FUNCTION_BLOCK FB_Observer_USINT EXTENDS FB_AbstractObserver
VAR
    _nVal:              USINT;
END_VAR

METHOD FB_init : BOOL
VAR_INPUT
	bInitRetains : BOOL; // if TRUE, the retain variables are initialized (warm start / cold start)
	bInCopyCode : BOOL;  // if TRUE, the instance afterwards gets moved into the copy code (online change)
END_VAR
THIS^._nTypeClass := __SYSTEM.TYPE_CLASS.TYPE_USINT;
THIS^._pVal := ADR(THIS^._nVal);
THIS^._nSize := SIZEOF(THIS^._nVal);
END_METHOD

PROPERTY nValue8 : USINT
GET
nValue8 := THIS^._nVal;
END_GET
END_PROPERTY

END_FUNCTION_BLOCK

(* stored: Version 1.1.0.1, ProductVersion 3.1.4024.12
   POU FB_Observer_USINT: Id {96585317-5966-06f8-0c4a-6dc99eae77ca}, SpecialFunc None
   Method FB_init: Id {65d03af9-c1b6-07a0-3f4d-56ccaa09f6e3}
   Property nValue8: Id {5a0f3ccb-ac73-0b71-035b-998fa35ef5d4}
   Get Get: Id {4b8d5a07-c9ed-0dba-24fd-86e823f4b302} *)
